// TIA Portal V16 export
// export: Created 2022-11-17T11:55:26.0485381Z, ExportSetting WithDefaults, DisplayName Totally Integrated Automation Portal, DisplayVersion V16 Update 6, DisplayName TIA Portal Version Control Interface, DisplayVersion V16 Update 2, DisplayName TIA Portal Openness, DisplayVersion V16 Update 6, DisplayName SINAMICS Startdrive Advanced, DisplayVersion V16 Update 5, DisplayName SINAMICS Startdrive G130, G150, S120, S150, SINAMICS MV, S210, DisplayVersion V16 Update 5, DisplayName SINAMICS Startdrive G110M, G120, G120C, G120D, G120P, G115D, DisplayVersion V16 Update 5, DisplayName STEP 7 Professional, DisplayVersion V16 Update 6, DisplayName STEP 7 Safety, DisplayVersion V16, DisplayName WinCC Advanced, DisplayVersion V16 Update 6
DATA_BLOCK "DB06_Clamp"   // DB6
{ S7_Optimized_Access := 'FALSE' }
AUTHOR : Robopac
VERSION : 0.0
// stored: AutoNumber false, IsOnlyStoredInLoadMemory false, IsWriteProtectedInAS false
   VAR RETAIN
      dbx0_0 : Bool := FALSE;   // Welder contrast upward
      dbx0_1 : Bool := FALSE;   // Welder contrast downward
      dbx0_2 : Bool := FALSE;   // Welder unit upward
      dbx0_3 : Bool := FALSE;   // Welder unit downward
      dbx0_4 : Bool := FALSE;
      dbx0_5 : Bool := FALSE;   // Film clamp upward
      dbx0_6 : Bool := FALSE;   // Film clamp downward
      dbx0_7 : Bool := FALSE;   // Welder and cut unit forward
      dbx1_0 : Bool := FALSE;   // Welder and cut unit backward
      dbx1_1 : Bool := FALSE;
      dbx1_2 : Bool := FALSE;
      dbx1_3 : Bool := FALSE;
      dbx1_4 : Bool := FALSE;
      dbx1_5 : Bool := FALSE;
      dbx1_6 : Bool := FALSE;
      dbx1_7 : Bool := FALSE;
      dbx2_0 : Bool := FALSE;   // Welder contrast forward
      dbx2_1 : Bool := FALSE;   // Welder contrast backward
      dbx2_2 : Bool := FALSE;
      dbx2_3 : Bool := FALSE;
      dbx2_4 : Bool := FALSE;
      dbx2_5 : Bool := FALSE;
      dbx2_6 : Bool := FALSE;
      dbx2_7 : Bool := FALSE;
      dbb3 : Byte := 16#00;
      dbx4_0 : Bool := FALSE;   // Spool carrage upward to cover tail
      dbx4_1 : Bool := FALSE;   // Spool carrage downward after film tail covered
      dbx4_2 : Bool := FALSE;   // Spool carrage upward at the begining
      dbx4_3 : Bool := FALSE;   // Spool carriage height to pull film at begining
      dbx4_4 : Bool := FALSE;   // Support memory for revolution over welder contrast
      dbx4_5 : Bool := TRUE;   // Clamp carriage is not backward because wrapping cycle
      dbb5 : Byte := 16#00;
      dbw6 : Int := 0;
      dbw8 : Int := 0;
      dbw10 : Int := 500;   // Spool carriage height for film tail airblower
      dbw12 : Int := 0;   // Number of revolution to open clamp
      dbw14 : Int := 0;   // Spool carriage height for film tail wrapped
      dbw16 : Int := 200;   // Spool carriage height to enable revolution over clamp
      dbw18 : Int := 1942;
      dbw20 : Int := 0;
      dbw22 : Int := 0;
      dbw24 : Int := 0;
      dbw26 : Int := 0;
      dbw28 : Int := 0;
      dbw30 : Int := 0;
      dbw32 : Int := 0;
      dbw34 : Int := 0;
      dbw36 : Int := 0;
      dbw38 : Int := 0;
      dbw40 : Int := 0;   // Delay to open clamp (number of 100msec)
      dbw42 : Int := 0;   // Time to open clamp related to actual speed
      dbw44 : Int := 0;
      dbw46 : Int := 0;
      dbw48 : Int := 0;
   END_VAR
BEGIN
END_DATA_BLOCK
